TYPE DUT_IO :
STRUCT
	I_isOpen: BOOL := FALSE;
	I_isClosed: BOOL := FALSE;
	I_hasFailure: BOOL := FALSE;
	O_setOpen: BOOL := FALSE;
END_STRUCT
END_TYPE

(* stored: Version 1.1.0.1, ProductVersion 3.1.4024.12
   DUT DUT_IO: Id {58cd96ab-b9f7-4ce1-bc12-5184398eafc7} *)
